TYPE Module_Palletizer_Aspirazione_ManCmd :
STRUCT
	AttivazioneVuoto 	: BOOL;
	DisattivazioneVuoto : BOOL;
	SalitaVentose		: BOOL;
	DiscesaVentose		: BOOL;
	Home				: BOOL;
END_STRUCT
END_TYPE

(* stored: Version 1.1.0.1, ProductVersion 3.1.4024.11
   DUT Module_Palletizer_Aspirazione_ManCmd: Id {c32d2ebe-c551-424f-9767-52eeee246fa4} *)
